// TwinCAT 3 PLC project PLC_workshop_SourceControl
// ProgramVersion: 3.1.4023.0
// libraries:
//   Tc2_Standard, * (Beckhoff Automation GmbH)
//   Tc2_System, * (Beckhoff Automation GmbH)
//   Tc3_Module, * (Beckhoff Automation GmbH)
// project tree:
//   / PlcTask.TcTTO
//   POUs/ MAIN.TcPOU, POU_LAD.TcPOU
// real-time tasks:
//   TASK PlcTask: cycle T#10ms, priority 20, ADS port 350

CONFIGURATION PLC_workshop_SourceControl
    RESOURCE PLC ON TwinCAT3
        TASK PlcTask(INTERVAL := T#10ms, PRIORITY := 20);
        PROGRAM MAIN WITH PlcTask : MAIN;
    END_RESOURCE
END_CONFIGURATION

// ---- POUs/MAIN.TcPOU
PROGRAM MAIN
VAR
	//cmt 1
	bTest_1 : BOOL;
	
	//cmt 2
	bTest_2 : BOOL;
END_VAR

// --- Version 1 --- 
// Program 1
// -----------------


// --- Version 2 --- 
// Program 2
// -----------------


// --- Version 3 --- 
// Khang
// -----------------

END_PROGRAM

// ---- POUs/POU_LAD.TcPOU
PROGRAM POU_LAD
VAR
	in_1	: BOOL;
	out_1	: BOOL;
END_VAR

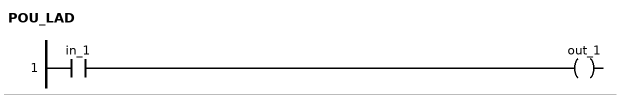
// NETWORK 1
out_1 := in_1;

END_PROGRAM
